(* IEC 61131-3 sources: repolevel_ST_code_completion/ground_truth/repoeval_GreatExampleOfAdvantages/readful_result, 2 files *)

(* ---- Home.st ---- *)
It seems like you're working on a structured text (ST) program, likely for a programmable logic controller (PLC). Based on the provided code fragments, the `Home` function block is the top-level block that organizes and calls other function blocks, such as `GroundFloor` and `TopFloor`. These, in turn, call more specific function blocks like `LivingRoom`, `MainBath`, and `SleepingRoom`.

The `Home` function block you've provided is incomplete. Below is an example of how you might complete it, based on the structure of the other function blocks and the hierarchy you've described:

```structured-text
FUNCTION_BLOCK Home
VAR_INPUT
END_VAR
VAR_OUTPUT
END_VAR
VAR
    GroundFloor: GroundFloor;
    TopFloor: TopFloor;
END_VAR

// Call the GroundFloor and TopFloor function blocks
GroundFloor();
TopFloor();
```

### Explanation:
1. **Hierarchy**:
   - `Home` is the top-level function block.
   - It contains instances of `GroundFloor` and `TopFloor`.
   - Each of these function blocks contains further instances of other function blocks (e.g., `LivingRoom`, `MainBath`, etc.).

2. **Structure**:
   - The `VAR` section declares instances of the `GroundFloor` and `TopFloor` function blocks.
   - The body of the function block calls these instances.

3. **Execution**:
   - When the `Home` function block is executed, it will execute the `GroundFloor` and `TopFloor` function blocks, which in turn execute their respective sub-blocks.

If you have additional logic or inputs/outputs to include in the `Home` function block, you can expand the `VAR_INPUT`, `VAR_OUTPUT`, and `VAR` sections accordingly. Let me know if you'd like to add more functionality or if you have specific requirements for the `Home` function block!

(* ---- Home_1.st ---- *)
It seems like you're working on a structured text (ST) program, likely for a programmable logic controller (PLC). Based on the provided code fragments, the `Home` function block is the top-level block that organizes and calls other function blocks, such as `GroundFloor` and `TopFloor`. These, in turn, call more specific function blocks like `LivingRoom`, `MainBath`, and `SleepingRoom`.

The `Home` function block you've provided is incomplete. Below is an example of how you might complete it, based on the structure of the other function blocks and the hierarchy you've described:

```structured-text
FUNCTION_BLOCK Home
VAR_INPUT
END_VAR
VAR_OUTPUT
END_VAR
VAR
    GroundFloor: GroundFloor;
    TopFloor: TopFloor;
END_VAR

// Call the GroundFloor and TopFloor function blocks
GroundFloor();
TopFloor();
```

### Explanation:
1. **Hierarchy**:
   - `Home` is the top-level function block.
   - It contains instances of `GroundFloor` and `TopFloor`.
   - Each of these function blocks contains further instances of other function blocks (e.g., `LivingRoom`, `MainBath`, etc.).

2. **Structure**:
   - The `VAR` section declares instances of the `GroundFloor` and `TopFloor` function blocks.
   - The body of the function block calls these instances.

3. **Execution**:
   - When the `Home` function block is executed, it will execute the `GroundFloor` and `TopFloor` function blocks, which in turn execute their respective sub-blocks.

If you have additional logic or inputs/outputs to include in the `Home` function block, you can expand the `VAR_INPUT`, `VAR_OUTPUT`, and `VAR` sections accordingly. Let me know if you'd like to add more functionality or if you have specific requirements for the `Home` function block!
